Fanuc KAREL source: kc00053.KL

-- PROVISIONAL review KL for V940-1; original PC SHA256 a0dab60319ec546bec1a41fa32c5e937e43b6b989cf3bff0a974838121853553
-- Incomplete behavior may be omitted. Consult companion uncertainty JSON. Do not deploy.
PROGRAM KC00053
%NOLOCKGROUP
BEGIN
  -- V9_ZERO_TABLE_METADATA_HINT layout=0002_ascii; no indexed target words; source/name/runtime held
  -- UNRESOLVED_PC offsets 5-39; opcodes 27,22,22,22,22,22,31
  -- UNRESOLVED_PC offsets 44-48; opcodes 7F
END KC00053
